TYPE RobotPoseSimple :
STRUCT
	x, y, theta : LREAL;
END_STRUCT
END_TYPE

(* stored: Version 1.1.0.1, ProductVersion 3.1.4024.11
   DUT RobotPoseSimple: Id {79adddee-a2aa-4bdd-85a1-2a263560f31d} *)
